TYPE "PPrf_CoilHandling_MaterialFeeding"
VERSION : 0.1
// Block: PPrf_CoilHandling_MaterialFeeding
   STRUCT
      DecoilerFeedMode : UInt;
      StraightenerRollsUse : UInt;
      Vel : LReal;
      Acc : LReal;
      Dec : LReal;
      Jerk : LReal;
   END_STRUCT;

END_TYPE
